// TIA Portal V18 export
FUNCTION "AObasic" : Void   // FC10002, FBD
{ S7_Optimized_Access := 'TRUE' }
VERSION : 0.1
// stored: AutoNumber false, IsIECCheckEnabled false, SetENOAutomatically false, UDAEnableTagReadback false
   VAR_INPUT
      rInput : Real;   // 0 to 100
      cM0A : Byte;   // 0-direct / 1-reverse / 0-outp_off / 1- out=MAN_OUTPUT /2 -out=input
      rManOutput : Real;
   END_VAR
   VAR_OUTPUT
      iOutput : Int;
   END_VAR
   VAR_TEMP
      rOut : Real;
      iOut : Int;
      rManOutputTemp : Real;
      iManOutputTemp : Int;
   END_VAR
BEGIN

REGION Network 1
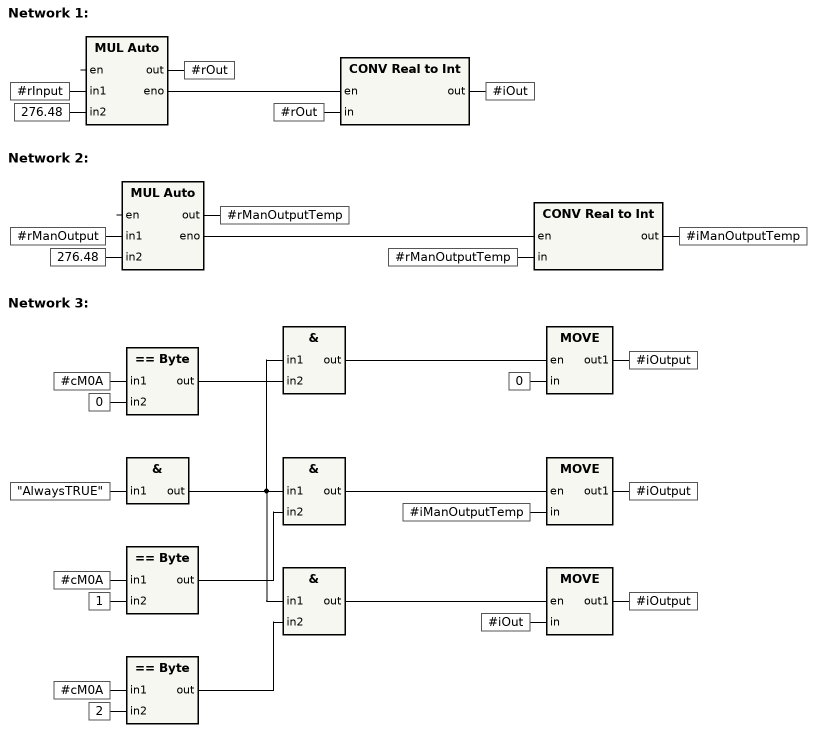
   #rOut := #rInput * 276.48;
   #iOut := REAL_TO_INT(#rOut);
END_REGION

REGION Network 2
   #rManOutputTemp := #rManOutput * 276.48;
   #iManOutputTemp := REAL_TO_INT(#rManOutputTemp);
END_REGION

REGION Network 3
   IF "AlwaysTRUE" AND (#cM0A = 0) THEN #iOutput := 0; END_IF;
   IF "AlwaysTRUE" AND (#cM0A = 1) THEN #iOutput := #iManOutputTemp; END_IF;
   IF "AlwaysTRUE" AND (#cM0A = 2) THEN #iOutput := #iOut; END_IF;
END_REGION
END_FUNCTION
